INTERFACE I_BaseElement EXTENDS I_Disposable, I_HaveContent, I_HaveInputPorts, I_HaveOutputPorts, I_HaveErrors, I_HaveProperties, I_HaveExtensions, I_HaveMetadata, I_EventEmitter, __SYSTEM.IQueryInterface

END_INTERFACE

(* stored: Version 1.1.0.1, ProductVersion 3.1.4024.12
   Itf I_BaseElement: Id {edccaa5e-b335-05b5-362b-cf76e03aa61c} *)
